Fanuc KAREL source: kt00161.KL

PROGRAM KT00161
%NOLOCKGROUP
VAR
I1:INTEGER;I2:INTEGER;OUT:INTEGER
BEGIN
--
--
I1=2
I2=3
I1=2
I2=3
OUT=(I1 MOD I2)
END KT00161
